INTERFACE I_Cam_Ctrl

PROPERTY Axes : reference TO ARRAY[1..PLC_CONSTANT.MAX_AXIS] OF AXIS_REF
SET
END_SET
END_PROPERTY

PROPERTY AxisCtrl : pointer to ARRAY[1..PLC_CONSTANT.MAX_AXIS] OF st_axis_ctrl
SET
END_SET
END_PROPERTY

PROPERTY AxisData : pointer to ARRAY[1..PLC_CONSTANT.MAX_AXIS] OF ST_CAM_DATA
SET
END_SET
END_PROPERTY

PROPERTY AxisIndex : uint
SET
END_SET
END_PROPERTY

PROPERTY AxisInfo : pointer to ARRAY[1..PLC_CONSTANT.MAX_AXIS] OF ST_AXIS_INFO
SET
END_SET
END_PROPERTY

PROPERTY AxisState : pointer to ARRAY[1..PLC_CONSTANT.MAX_AXIS] OF ST_CAM_STATE
SET
END_SET
END_PROPERTY

METHOD Cycle  : e_progress
END_METHOD

PROPERTY ItfMcAxes : array[1..MAX_AXIS] of I_McAxis
SET
END_SET
END_PROPERTY

PROPERTY MessageLevel : E_MessageType
SET
END_SET
END_PROPERTY

PROPERTY MotionFunction : POINTER TO ARRAY[1..MAX_AXIS] OF ST_MOTION_FUNCTION
SET
END_SET
END_PROPERTY

PROPERTY MotionFunctionPoint : pointer to array[1..MAX_AXIS] of ST_MOTION_FUNCTION_POINT
SET
END_SET
END_PROPERTY

END_INTERFACE

(* stored: Version 1.1.0.1, ProductVersion 3.1.4024.12
   Itf I_Cam_Ctrl: Id {4e1da497-37ee-0168-2b24-5b9fbd7bcd6c}
   Folder methods: Id {289023ab-c939-0f43-2a6d-f07aa32fae6f}
   Folder properties: Id {b935bae4-20b3-043e-188d-a7ce7fdbdbf3}
   Property Axes: Id {8193c79d-7247-0d2a-310f-9467f21399fd}
   Set Set: Id {2c47bb15-1372-0be6-0216-0353b4106f86}
   Property AxisCtrl: Id {b628aab6-43ad-06cd-37b3-8ef1894d8490}
   Set Set: Id {ab5a31ec-2c82-0876-0f62-23ae259eabe0}
   Property AxisData: Id {29e79334-8275-0433-3468-1bd12dc7b2a9}
   Set Set: Id {66951bb9-3ec4-042a-108a-c31f69b5b650}
   Property AxisIndex: Id {62db2c89-35b0-0068-2019-ab74ffbaf9ec}
   Set Set: Id {0083986f-5ddb-0d8f-1af0-45885d80f1f2}
   Property AxisInfo: Id {c4e78251-8097-003e-3bad-03f58172a569}
   Set Set: Id {5cb24616-3f31-0aff-1029-27202044ad6a}
   Property AxisState: Id {b3fad775-854f-0465-13df-2a6b7819623a}
   Set Set: Id {f00d57f8-9c0c-0ddd-2468-d15ea26ab47d}
   Method Cycle: Id {ce9f2a1e-2df8-0349-1e51-54c4c0c7254a}
   Property ItfMcAxes: Id {9c279bcc-d788-0eae-035d-8ae9b3fba035}
   Set Set: Id {9f1667da-a83f-0010-2d1e-715bceceb278}
   Property MessageLevel: Id {fd50ea6d-ea07-021c-1a8b-ab91ef8e6039}
   Set Set: Id {d67756da-c6a8-0d9e-1c52-24998f70935d}
   Property MotionFunction: Id {51497f92-2c5d-0340-36c3-d2c881e7309b}
   Set Set: Id {87417229-730c-082b-137d-28ee01332c1d}
   Property MotionFunctionPoint: Id {3ccce8b0-462d-0c84-1a27-b7acfc79c954}
   Set Set: Id {8a11a43b-80fd-00e4-0e64-27354f449965} *)
